FUNCTION_BLOCK Imshow (* openCV show image *)
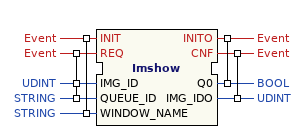
  EVENT_INPUT
    INIT WITH WINDOW_NAME;
    REQ WITH IMG_ID, QUEUE_ID;
  END_EVENT
  EVENT_OUTPUT
    INITO WITH Q0;
    CNF WITH IMG_IDO;
  END_EVENT
  VAR_INPUT
    IMG_ID : UDINT;
    QUEUE_ID : STRING;
    WINDOW_NAME : STRING;
  END_VAR
  VAR_OUTPUT
    Q0 : BOOL;
    IMG_IDO : UDINT;
  END_VAR
END_FUNCTION_BLOCK
